  650 = 'Clamp Cylinder A1 Failed to Advance... Check Q1.0...' | German: 'S3 650 Row 66 Failed To Advance.. Check Qxxx.x German' | French: 'S3 650 Row 66 Failed To Advance.. Check Qxxx.x French'
  651 = 'Clamp Cylinder A1 Failed to Return... Check Q1.1...' | German: 'S3 651 Row 66 Failed To Return.. Check Qxxx.x German' | French: 'S3 651 Row 66 Failed To Return.. Check Qxxx.x French'
  652 = 'Clamp Cylinder A1 Lost Advanced... Check I1.0...' | German: 'S3 652 Row 66 Lost Advance Position... Check Ixxx.x German' | French: 'S3 652 Row 66 Lost Advance Position... Check Ixxx.x French'
  653 = 'Clamp Cylinder A1 Lost Returned... Check I1.1...' | German: 'S3 653 Row 66 Lost Return Position... Check Ixxx.x German' | French: 'S3 653 Row 66 Lost Return Position... Check Ixxx.x French'
  654 = 'Clamp Cylinder A1 Switch Fault... Check I1.0, I1.1...' | German: 'S3 654 Row 66 Switch Fault... Check Ixxx.x / Ixxx.x German' | French: 'S3 654 Row 66 Switch Fault... Check Ixxx.x / Ixxx.x French'
  655 = 'Spare' | German: 'S3 655 Row 66 Spare Message German' | French: 'S3 655 Row 66 Spare Message French'
  656 = 'Spare' | German: 'S3 656 Row 66 Spare Message German' | French: 'S3 656 Row 66 Spare Message French'
  657 = 'Spare' | German: 'S3 657 Row 66 Spare Message German' | French: 'S3 657 Row 66 Spare Message French'
  658 = 'Spare' | German: 'S3 658 Row 66 Spare Message German' | French: 'S3 658 Row 66 Spare Message French'
  659 = 'Spare' | German: 'S3 659 Row 66 Spare Message German' | French: 'S3 659 Row 66 Spare Message French'
  660 = 'Clamp Cylinder A1 Failed to Advance... Check Q1.0...' | German: 'S3 660 Row 67 Failed To Advance.. Check Qxxx.x German' | French: 'S3 660 Row 67 Failed To Advance.. Check Qxxx.x French'
  661 = 'Clamp Cylinder A1 Failed to Return... Check Q1.1...' | German: 'S3 661 Row 67 Failed To Return.. Check Qxxx.x German' | French: 'S3 661 Row 67 Failed To Return.. Check Qxxx.x French'
  662 = 'Clamp Cylinder A1 Lost Advanced... Check I1.0...' | German: 'S3 662 Row 67 Lost Advance Position... Check Ixxx.x German' | French: 'S3 662 Row 67 Lost Advance Position... Check Ixxx.x French'
  663 = 'Clamp Cylinder A1 Lost Returned... Check I1.1...' | German: 'S3 663 Row 67 Lost Return Position... Check Ixxx.x German' | French: 'S3 663 Row 67 Lost Return Position... Check Ixxx.x French'
  664 = 'Clamp Cylinder A1 Switch Fault... Check I1.0, I1.1...' | German: 'S3 664 Row 67 Switch Fault... Check Ixxx.x / Ixxx.x German' | French: 'S3 664 Row 67 Switch Fault... Check Ixxx.x / Ixxx.x French'
  665 = 'Spare' | German: 'S3 665 Row 67 Spare Message German' | French: 'S3 665 Row 67 Spare Message French'
  666 = 'Spare' | German: 'S3 666 Row 67 Spare Message German' | French: 'S3 666 Row 67 Spare Message French'
  667 = 'Spare' | German: 'S3 667 Row 67 Spare Message German' | French: 'S3 667 Row 67 Spare Message French'
  668 = 'Spare' | German: 'S3 668 Row 67 Spare Message German' | French: 'S3 668 Row 67 Spare Message French'
  669 = 'Spare' | German: 'S3 669 Row 67 Spare Message German' | French: 'S3 669 Row 67 Spare Message French'
  670 = 'Clamp Cylinder A1 Failed to Advance... Check Q1.0...' | German: 'S3 670 Row 68 Failed To Advance.. Check Qxxx.x German' | French: 'S3 670 Row 68 Failed To Advance.. Check Qxxx.x French'
  671 = 'Clamp Cylinder A1 Failed to Return... Check Q1.1...' | German: 'S3 671 Row 68 Failed To Return.. Check Qxxx.x German' | French: 'S3 671 Row 68 Failed To Return.. Check Qxxx.x French'
  672 = 'Clamp Cylinder A1 Lost Advanced... Check I1.0...' | German: 'S3 672 Row 68 Lost Advance Position... Check Ixxx.x German' | French: 'S3 672 Row 68 Lost Advance Position... Check Ixxx.x French'
  673 = 'Clamp Cylinder A1 Lost Returned... Check I1.1...' | German: 'S3 673 Row 68 Lost Return Position... Check Ixxx.x German' | French: 'S3 673 Row 68 Lost Return Position... Check Ixxx.x French'
  674 = 'Clamp Cylinder A1 Switch Fault... Check I1.0, I1.1...' | German: 'S3 674 Row 68 Switch Fault... Check Ixxx.x / Ixxx.x German' | French: 'S3 674 Row 68 Switch Fault... Check Ixxx.x / Ixxx.x French'
  675 = 'Spare' | German: 'S3 675 Row 68 Spare Message German' | French: 'S3 675 Row 68 Spare Message French'
  676 = 'Spare' | German: 'S3 676 Row 68 Spare Message German' | French: 'S3 676 Row 68 Spare Message French'
  677 = 'Spare' | German: 'S3 677 Row 68 Spare Message German' | French: 'S3 677 Row 68 Spare Message French'
  678 = 'Spare' | German: 'S3 678 Row 68 Spare Message German' | French: 'S3 678 Row 68 Spare Message French'
  679 = 'Spare' | German: 'S3 679 Row 68 Spare Message German' | French: 'S3 679 Row 68 Spare Message French'
  680 = 'Clamp Cylinder A1 Failed to Advance... Check Q1.0...' | German: 'S3 680 Row 69 Failed To Advance.. Check Qxxx.x German' | French: 'S3 680 Row 69 Failed To Advance.. Check Qxxx.x French'
  681 = 'Clamp Cylinder A1 Failed to Return... Check Q1.1...' | German: 'S3 681 Row 69 Failed To Return.. Check Qxxx.x German' | French: 'S3 681 Row 69 Failed To Return.. Check Qxxx.x French'
  682 = 'Clamp Cylinder A1 Lost Advanced... Check I1.0...' | German: 'S3 682 Row 69 Lost Advance Position... Check Ixxx.x German' | French: 'S3 682 Row 69 Lost Advance Position... Check Ixxx.x French'
  683 = 'Clamp Cylinder A1 Lost Returned... Check I1.1...' | German: 'S3 683 Row 69 Lost Return Position... Check Ixxx.x German' | French: 'S3 683 Row 69 Lost Return Position... Check Ixxx.x French'
  684 = 'Clamp Cylinder A1 Switch Fault... Check I1.0, I1.1...' | German: 'S3 684 Row 69 Switch Fault... Check Ixxx.x / Ixxx.x German' | French: 'S3 684 Row 69 Switch Fault... Check Ixxx.x / Ixxx.x French'
  685 = 'Spare' | German: 'S3 685 Row 69 Spare Message German' | French: 'S3 685 Row 69 Spare Message French'
  686 = 'Spare' | German: 'S3 686 Row 69 Spare Message German' | French: 'S3 686 Row 69 Spare Message French'
  687 = 'Spare' | German: 'S3 687 Row 69 Spare Message German' | French: 'S3 687 Row 69 Spare Message French'
  688 = 'Spare' | German: 'S3 688 Row 69 Spare Message German' | French: 'S3 688 Row 69 Spare Message French'
  689 = 'Spare' | German: 'S3 689 Row 69 Spare Message German' | French: 'S3 689 Row 69 Spare Message French'
  690 = 'Clamp Cylinder A1 Failed to Advance... Check Q1.0...' | German: 'S3 690 Row 70 Failed To Advance.. Check Qxxx.x German' | French: 'S3 690 Row 70 Failed To Advance.. Check Qxxx.x French'
  691 = 'Clamp Cylinder A1 Failed to Return... Check Q1.1...' | German: 'S3 691 Row 70 Failed To Return.. Check Qxxx.x German' | French: 'S3 691 Row 70 Failed To Return.. Check Qxxx.x French'
  692 = 'Clamp Cylinder A1 Lost Advanced... Check I1.0...' | German: 'S3 692 Row 70 Lost Advance Position... Check Ixxx.x German' | French: 'S3 692 Row 70 Lost Advance Position... Check Ixxx.x French'
  693 = 'Clamp Cylinder A1 Lost Returned... Check I1.1...' | German: 'S3 693 Row 70 Lost Return Position... Check Ixxx.x German' | French: 'S3 693 Row 70 Lost Return Position... Check Ixxx.x French'
  694 = 'Clamp Cylinder A1 Switch Fault... Check I1.0, I1.1...' | German: 'S3 694 Row 70 Switch Fault... Check Ixxx.x / Ixxx.x German' | French: 'S3 694 Row 70 Switch Fault... Check Ixxx.x / Ixxx.x French'
  695 = 'Spare' | German: 'S3 695 Row 70 Spare Message German' | French: 'S3 695 Row 70 Spare Message French'
  696 = 'Spare' | German: 'S3 696 Row 70 Spare Message German' | French: 'S3 696 Row 70 Spare Message French'
  697 = 'Spare' | German: 'S3 697 Row 70 Spare Message German' | French: 'S3 697 Row 70 Spare Message French'
  698 = 'Spare' | German: 'S3 698 Row 70 Spare Message German' | French: 'S3 698 Row 70 Spare Message French'
  699 = 'Spare' | German: 'S3 699 Row 70 Spare Message German' | French: 'S3 699 Row 70 Spare Message French'
  700 = 'Clamp Cylinder A1 Failed to Advance... Check Q1.0...' | German: 'S3 700 Row 71 Failed To Advance.. Check Qxxx.x German' | French: 'S3 700 Row 71 Failed To Advance.. Check Qxxx.x French'
  701 = 'Clamp Cylinder A1 Failed to Return... Check Q1.1...' | German: 'S3 701 Row 71 Failed To Return.. Check Qxxx.x German' | French: 'S3 701 Row 71 Failed To Return.. Check Qxxx.x French'
  702 = 'Clamp Cylinder A1 Lost Advanced... Check I1.0...' | German: 'S3 702 Row 71 Lost Advance Position... Check Ixxx.x German' | French: 'S3 702 Row 71 Lost Advance Position... Check Ixxx.x French'
  703 = 'Clamp Cylinder A1 Lost Returned... Check I1.1...' | German: 'S3 703 Row 71 Lost Return Position... Check Ixxx.x German' | French: 'S3 703 Row 71 Lost Return Position... Check Ixxx.x French'
  704 = 'Clamp Cylinder A1 Switch Fault... Check I1.0, I1.1...' | German: 'S3 704 Row 71 Switch Fault... Check Ixxx.x / Ixxx.x German' | French: 'S3 704 Row 71 Switch Fault... Check Ixxx.x / Ixxx.x French'
  705 = 'Spare' | German: 'S3 705 Row 71 Spare Message German' | French: 'S3 705 Row 71 Spare Message French'
  706 = 'Spare' | German: 'S3 706 Row 71 Spare Message German' | French: 'S3 706 Row 71 Spare Message French'
  707 = 'Spare' | German: 'S3 707 Row 71 Spare Message German' | French: 'S3 707 Row 71 Spare Message French'
  708 = 'Spare' | German: 'S3 708 Row 71 Spare Message German' | French: 'S3 708 Row 71 Spare Message French'
  709 = 'Spare' | German: 'S3 709 Row 71 Spare Message German' | French: 'S3 709 Row 71 Spare Message French'
  710 = 'Clamp Cylinder A1 Failed to Advance... Check Q1.0...' | German: 'S3 710 Row 72 Failed To Advance.. Check Qxxx.x German' | French: 'S3 710 Row 72 Failed To Advance.. Check Qxxx.x French'
  711 = 'Clamp Cylinder A1 Failed to Return... Check Q1.1...' | German: 'S3 711 Row 72 Failed To Return.. Check Qxxx.x German' | French: 'S3 711 Row 72 Failed To Return.. Check Qxxx.x French'
  712 = 'Clamp Cylinder A1 Lost Advanced... Check I1.0...' | German: 'S3 712 Row 72 Lost Advance Position... Check Ixxx.x German' | French: 'S3 712 Row 72 Lost Advance Position... Check Ixxx.x French'
  713 = 'Clamp Cylinder A1 Lost Returned... Check I1.1...' | German: 'S3 713 Row 72 Lost Return Position... Check Ixxx.x German' | French: 'S3 713 Row 72 Lost Return Position... Check Ixxx.x French'
  714 = 'Clamp Cylinder A1 Switch Fault... Check I1.0, I1.1...' | German: 'S3 714 Row 72 Switch Fault... Check Ixxx.x / Ixxx.x German' | French: 'S3 714 Row 72 Switch Fault... Check Ixxx.x / Ixxx.x French'
  715 = 'Spare' | German: 'S3 715 Row 72 Spare Message German' | French: 'S3 715 Row 72 Spare Message French'
  716 = 'Spare' | German: 'S3 716 Row 72 Spare Message German' | French: 'S3 716 Row 72 Spare Message French'
  717 = 'Spare' | German: 'S3 717 Row 72 Spare Message German' | French: 'S3 717 Row 72 Spare Message French'
  718 = 'Spare' | German: 'S3 718 Row 72 Spare Message German' | French: 'S3 718 Row 72 Spare Message French'
  719 = 'Spare' | German: 'S3 719 Row 72 Spare Message German' | French: 'S3 719 Row 72 Spare Message French'
  720 = 'Clamp Cylinder A1 Failed to Advance... Check Q1.0...' | German: 'S3 720 Row 73 Failed To Advance.. Check Qxxx.x German' | French: 'S3 720 Row 73 Failed To Advance.. Check Qxxx.x French'
  721 = 'Clamp Cylinder A1 Failed to Return... Check Q1.1...' | German: 'S3 721 Row 73 Failed To Return.. Check Qxxx.x German' | French: 'S3 721 Row 73 Failed To Return.. Check Qxxx.x French'
  722 = 'Clamp Cylinder A1 Lost Advanced... Check I1.0...' | German: 'S3 722 Row 73 Lost Advance Position... Check Ixxx.x German' | French: 'S3 722 Row 73 Lost Advance Position... Check Ixxx.x French'
  723 = 'Clamp Cylinder A1 Lost Returned... Check I1.1...' | German: 'S3 723 Row 73 Lost Return Position... Check Ixxx.x German' | French: 'S3 723 Row 73 Lost Return Position... Check Ixxx.x French'
  724 = 'Clamp Cylinder A1 Switch Fault... Check I1.0, I1.1...' | German: 'S3 724 Row 73 Switch Fault... Check Ixxx.x / Ixxx.x German' | French: 'S3 724 Row 73 Switch Fault... Check Ixxx.x / Ixxx.x French'
  725 = 'Spare' | German: 'S3 725 Row 73 Spare Message German' | French: 'S3 725 Row 73 Spare Message French'
  726 = 'Spare' | German: 'S3 726 Row 73 Spare Message German' | French: 'S3 726 Row 73 Spare Message French'
  727 = 'Spare' | German: 'S3 727 Row 73 Spare Message German' | French: 'S3 727 Row 73 Spare Message French'
  728 = 'Spare' | German: 'S3 728 Row 73 Spare Message German' | French: 'S3 728 Row 73 Spare Message French'
  729 = 'Spare' | German: 'S3 729 Row 73 Spare Message German' | French: 'S3 729 Row 73 Spare Message French'
  730 = 'Clamp Cylinder A1 Failed to Advance... Check Q1.0...' | German: 'S3 730 Row 74 Failed To Advance.. Check Qxxx.x German' | French: 'S3 730 Row 74 Failed To Advance.. Check Qxxx.x French'
  731 = 'Clamp Cylinder A1 Failed to Return... Check Q1.1...' | German: 'S3 731 Row 74 Failed To Return.. Check Qxxx.x German' | French: 'S3 731 Row 74 Failed To Return.. Check Qxxx.x French'
  732 = 'Clamp Cylinder A1 Lost Advanced... Check I1.0...' | German: 'S3 732 Row 74 Lost Advance Position... Check Ixxx.x German' | French: 'S3 732 Row 74 Lost Advance Position... Check Ixxx.x French'
  733 = 'Clamp Cylinder A1 Lost Returned... Check I1.1...' | German: 'S3 733 Row 74 Lost Return Position... Check Ixxx.x German' | French: 'S3 733 Row 74 Lost Return Position... Check Ixxx.x French'
  734 = 'Clamp Cylinder A1 Switch Fault... Check I1.0, I1.1...' | German: 'S3 734 Row 74 Switch Fault... Check Ixxx.x / Ixxx.x German' | French: 'S3 734 Row 74 Switch Fault... Check Ixxx.x / Ixxx.x French'
  735 = 'Spare' | German: 'S3 735 Row 74 Spare Message German' | French: 'S3 735 Row 74 Spare Message French'
  736 = 'Spare' | German: 'S3 736 Row 74 Spare Message German' | French: 'S3 736 Row 74 Spare Message French'
  737 = 'Spare' | German: 'S3 737 Row 74 Spare Message German' | French: 'S3 737 Row 74 Spare Message French'
  738 = 'Spare' | German: 'S3 738 Row 74 Spare Message German' | French: 'S3 738 Row 74 Spare Message French'
  739 = 'Spare' | German: 'S3 739 Row 74 Spare Message German' | French: 'S3 739 Row 74 Spare Message French'
  740 = 'Clamp Cylinder A1 Failed to Advance... Check Q1.0...' | German: 'S3 740 Row 75 Failed To Advance.. Check Qxxx.x German' | French: 'S3 740 Row 75 Failed To Advance.. Check Qxxx.x French'
  741 = 'Clamp Cylinder A1 Failed to Return... Check Q1.1...' | German: 'S3 741 Row 75 Failed To Return.. Check Qxxx.x German' | French: 'S3 741 Row 75 Failed To Return.. Check Qxxx.x French'
  742 = 'Clamp Cylinder A1 Lost Advanced... Check I1.0...' | German: 'S3 742 Row 75 Lost Advance Position... Check Ixxx.x German' | French: 'S3 742 Row 75 Lost Advance Position... Check Ixxx.x French'
  743 = 'Clamp Cylinder A1 Lost Returned... Check I1.1...' | German: 'S3 743 Row 75 Lost Return Position... Check Ixxx.x German' | French: 'S3 743 Row 75 Lost Return Position... Check Ixxx.x French'
  744 = 'Clamp Cylinder A1 Switch Fault... Check I1.0, I1.1...' | German: 'S3 744 Row 75 Switch Fault... Check Ixxx.x / Ixxx.x German' | French: 'S3 744 Row 75 Switch Fault... Check Ixxx.x / Ixxx.x French'
  745 = 'Spare' | German: 'S3 745 Row 75 Spare Message German' | French: 'S3 745 Row 75 Spare Message French'
  746 = 'Spare' | German: 'S3 746 Row 75 Spare Message German' | French: 'S3 746 Row 75 Spare Message French'
  747 = 'Spare' | German: 'S3 747 Row 75 Spare Message German' | French: 'S3 747 Row 75 Spare Message French'
  748 = 'Spare' | German: 'S3 748 Row 75 Spare Message German' | French: 'S3 748 Row 75 Spare Message French'
  749 = 'Spare' | German: 'S3 749 Row 75 Spare Message German' | French: 'S3 749 Row 75 Spare Message French'
  750 = 'Clamp Cylinder A1 Failed to Advance... Check Q1.0...' | German: 'S3 750 Row 76 Failed To Advance.. Check Qxxx.x German' | French: 'S3 750 Row 76 Failed To Advance.. Check Qxxx.x French'
  751 = 'Clamp Cylinder A1 Failed to Return... Check Q1.1...' | German: 'S3 751 Row 76 Failed To Return.. Check Qxxx.x German' | French: 'S3 751 Row 76 Failed To Return.. Check Qxxx.x French'
  752 = 'Clamp Cylinder A1 Lost Advanced... Check I1.0...' | German: 'S3 752 Row 76 Lost Advance Position... Check Ixxx.x German' | French: 'S3 752 Row 76 Lost Advance Position... Check Ixxx.x French'
  753 = 'Clamp Cylinder A1 Lost Returned... Check I1.1...' | German: 'S3 753 Row 76 Lost Return Position... Check Ixxx.x German' | French: 'S3 753 Row 76 Lost Return Position... Check Ixxx.x French'
  754 = 'Clamp Cylinder A1 Switch Fault... Check I1.0, I1.1...' | German: 'S3 754 Row 76 Switch Fault... Check Ixxx.x / Ixxx.x German' | French: 'S3 754 Row 76 Switch Fault... Check Ixxx.x / Ixxx.x French'
  755 = 'Spare' | German: 'S3 755 Row 76 Spare Message German' | French: 'S3 755 Row 76 Spare Message French'
  756 = 'Spare' | German: 'S3 756 Row 76 Spare Message German' | French: 'S3 756 Row 76 Spare Message French'
  757 = 'Spare' | German: 'S3 757 Row 76 Spare Message German' | French: 'S3 757 Row 76 Spare Message French'
  758 = 'Spare' | German: 'S3 758 Row 76 Spare Message German' | French: 'S3 758 Row 76 Spare Message French'
  759 = 'Spare' | German: 'S3 759 Row 76 Spare Message German' | French: 'S3 759 Row 76 Spare Message French'
  760 = 'Clamp Cylinder A1 Failed to Advance... Check Q1.0...' | German: 'S3 760 Row 77 Failed To Advance.. Check Qxxx.x German' | French: 'S3 760 Row 77 Failed To Advance.. Check Qxxx.x French'
  761 = 'Clamp Cylinder A1 Failed to Return... Check Q1.1...' | German: 'S3 761 Row 77 Failed To Return.. Check Qxxx.x German' | French: 'S3 761 Row 77 Failed To Return.. Check Qxxx.x French'
  762 = 'Clamp Cylinder A1 Lost Advanced... Check I1.0...' | German: 'S3 762 Row 77 Lost Advance Position... Check Ixxx.x German' | French: 'S3 762 Row 77 Lost Advance Position... Check Ixxx.x French'
  763 = 'Clamp Cylinder A1 Lost Returned... Check I1.1...' | German: 'S3 763 Row 77 Lost Return Position... Check Ixxx.x German' | French: 'S3 763 Row 77 Lost Return Position... Check Ixxx.x French'
  764 = 'Clamp Cylinder A1 Switch Fault... Check I1.0, I1.1...' | German: 'S3 764 Row 77 Switch Fault... Check Ixxx.x / Ixxx.x German' | French: 'S3 764 Row 77 Switch Fault... Check Ixxx.x / Ixxx.x French'
  765 = 'Spare' | German: 'S3 765 Row 77 Spare Message German' | French: 'S3 765 Row 77 Spare Message French'
  766 = 'Spare' | German: 'S3 766 Row 77 Spare Message German' | French: 'S3 766 Row 77 Spare Message French'
  767 = 'Spare' | German: 'S3 767 Row 77 Spare Message German' | French: 'S3 767 Row 77 Spare Message French'
  768 = 'Spare' | German: 'S3 768 Row 77 Spare Message German' | French: 'S3 768 Row 77 Spare Message French'
  769 = 'Spare' | German: 'S3 769 Row 77 Spare Message German' | French: 'S3 769 Row 77 Spare Message French'
  770 = 'Clamp Cylinder A1 Failed to Advance... Check Q1.0...' | German: 'S3 770 Row 78 Failed To Advance.. Check Qxxx.x German' | French: 'S3 770 Row 78 Failed To Advance.. Check Qxxx.x French'
  771 = 'Clamp Cylinder A1 Failed to Return... Check Q1.1...' | German: 'S3 771 Row 78 Failed To Return.. Check Qxxx.x German' | French: 'S3 771 Row 78 Failed To Return.. Check Qxxx.x French'
  772 = 'Clamp Cylinder A1 Lost Advanced... Check I1.0...' | German: 'S3 772 Row 78 Lost Advance Position... Check Ixxx.x German' | French: 'S3 772 Row 78 Lost Advance Position... Check Ixxx.x French'
  773 = 'Clamp Cylinder A1 Lost Returned... Check I1.1...' | German: 'S3 773 Row 78 Lost Return Position... Check Ixxx.x German' | French: 'S3 773 Row 78 Lost Return Position... Check Ixxx.x French'
  774 = 'Clamp Cylinder A1 Switch Fault... Check I1.0, I1.1...' | German: 'S3 774 Row 78 Switch Fault... Check Ixxx.x / Ixxx.x German' | French: 'S3 774 Row 78 Switch Fault... Check Ixxx.x / Ixxx.x French'
  775 = 'Spare' | German: 'S3 775 Row 78 Spare Message German' | French: 'S3 775 Row 78 Spare Message French'
  776 = 'Spare' | German: 'S3 776 Row 78 Spare Message German' | French: 'S3 776 Row 78 Spare Message French'
  777 = 'Spare' | German: 'S3 777 Row 78 Spare Message German' | French: 'S3 777 Row 78 Spare Message French'
  778 = 'Spare' | German: 'S3 778 Row 78 Spare Message German' | French: 'S3 778 Row 78 Spare Message French'
  779 = 'Spare' | German: 'S3 779 Row 78 Spare Message German' | French: 'S3 779 Row 78 Spare Message French'
  780 = 'Clamp Cylinder A1 Failed to Advance... Check Q1.0...' | German: 'S3 780 Row 79 Failed To Advance.. Check Qxxx.x German' | French: 'S3 780 Row 79 Failed To Advance.. Check Qxxx.x French'
  781 = 'Clamp Cylinder A1 Failed to Return... Check Q1.1...' | German: 'S3 781 Row 79 Failed To Return.. Check Qxxx.x German' | French: 'S3 781 Row 79 Failed To Return.. Check Qxxx.x French'
  782 = 'Clamp Cylinder A1 Lost Advanced... Check I1.0...' | German: 'S3 782 Row 79 Lost Advance Position... Check Ixxx.x German' | French: 'S3 782 Row 79 Lost Advance Position... Check Ixxx.x French'
  783 = 'Clamp Cylinder A1 Lost Returned... Check I1.1...' | German: 'S3 783 Row 79 Lost Return Position... Check Ixxx.x German' | French: 'S3 783 Row 79 Lost Return Position... Check Ixxx.x French'
  784 = 'Clamp Cylinder A1 Switch Fault... Check I1.0, I1.1...' | German: 'S3 784 Row 79 Switch Fault... Check Ixxx.x / Ixxx.x German' | French: 'S3 784 Row 79 Switch Fault... Check Ixxx.x / Ixxx.x French'
  785 = 'Spare' | German: 'S3 785 Row 79 Spare Message German' | French: 'S3 785 Row 79 Spare Message French'
  786 = 'Spare' | German: 'S3 786 Row 79 Spare Message German' | French: 'S3 786 Row 79 Spare Message French'
  787 = 'Spare' | German: 'S3 787 Row 79 Spare Message German' | French: 'S3 787 Row 79 Spare Message French'
  788 = 'Spare' | German: 'S3 788 Row 79 Spare Message German' | French: 'S3 788 Row 79 Spare Message French'
  789 = 'Spare' | German: 'S3 789 Row 79 Spare Message German' | French: 'S3 789 Row 79 Spare Message French'
  790 = 'Clamp Cylinder A1 Failed to Advance... Check Q1.0...' | German: 'S3 790 Row 80 Failed To Advance.. Check Qxxx.x German' | French: 'S3 790 Row 80 Failed To Advance.. Check Qxxx.x French'
  791 = 'Clamp Cylinder A1 Failed to Return... Check Q1.1...' | German: 'S3 791 Row 80 Failed To Return.. Check Qxxx.x German' | French: 'S3 791 Row 80 Failed To Return.. Check Qxxx.x French'
  792 = 'Clamp Cylinder A1 Lost Advanced... Check I1.0...' | German: 'S3 792 Row 80 Lost Advance Position... Check Ixxx.x German' | French: 'S3 792 Row 80 Lost Advance Position... Check Ixxx.x French'
  793 = 'Clamp Cylinder A1 Lost Returned... Check I1.1...' | German: 'S3 793 Row 80 Lost Return Position... Check Ixxx.x German' | French: 'S3 793 Row 80 Lost Return Position... Check Ixxx.x French'
  794 = 'Clamp Cylinder A1 Switch Fault... Check I1.0, I1.1...' | German: 'S3 794 Row 80 Switch Fault... Check Ixxx.x / Ixxx.x German' | French: 'S3 794 Row 80 Switch Fault... Check Ixxx.x / Ixxx.x French'
  795 = 'Spare' | German: 'S3 795 Row 80 Spare Message German' | French: 'S3 795 Row 80 Spare Message French'
  796 = 'Spare' | German: 'S3 796 Row 80 Spare Message German' | French: 'S3 796 Row 80 Spare Message French'
  797 = 'Spare' | German: 'S3 797 Row 80 Spare Message German' | French: 'S3 797 Row 80 Spare Message French'
  798 = 'Spare' | German: 'S3 798 Row 80 Spare Message German' | French: 'S3 798 Row 80 Spare Message French'
  799 = 'Spare' | German: 'S3 799 Row 80 Spare Message German' | French: 'S3 799 Row 80 Spare Message French'
  800 = 'Clamp Cylinder A1 Failed to Advance... Check Q1.0...' | German: 'S3 800 Row 81 Failed To Advance.. Check Qxxx.x German' | French: 'S3 800 Row 81 Failed To Advance.. Check Qxxx.x French'
  801 = 'Clamp Cylinder A1 Failed to Return... Check Q1.1...' | German: 'S3 801 Row 81 Failed To Return.. Check Qxxx.x German' | French: 'S3 801 Row 81 Failed To Return.. Check Qxxx.x French'
  802 = 'Clamp Cylinder A1 Lost Advanced... Check I1.0...' | German: 'S3 802 Row 81 Lost Advance Position... Check Ixxx.x German' | French: 'S3 802 Row 81 Lost Advance Position... Check Ixxx.x French'
  803 = 'Clamp Cylinder A1 Lost Returned... Check I1.1...' | German: 'S3 803 Row 81 Lost Return Position... Check Ixxx.x German' | French: 'S3 803 Row 81 Lost Return Position... Check Ixxx.x French'
  804 = 'Clamp Cylinder A1 Switch Fault... Check I1.0, I1.1...' | German: 'S3 804 Row 81 Switch Fault... Check Ixxx.x / Ixxx.x German' | French: 'S3 804 Row 81 Switch Fault... Check Ixxx.x / Ixxx.x French'
  805 = 'Spare' | German: 'S3 805 Row 81 Spare Message German' | French: 'S3 805 Row 81 Spare Message French'
  806 = 'Spare' | German: 'S3 806 Row 81 Spare Message German' | French: 'S3 806 Row 81 Spare Message French'
  807 = 'Spare' | German: 'S3 807 Row 81 Spare Message German' | French: 'S3 807 Row 81 Spare Message French'
  808 = 'Spare' | German: 'S3 808 Row 81 Spare Message German' | French: 'S3 808 Row 81 Spare Message French'
  809 = 'Spare' | German: 'S3 809 Row 81 Spare Message German' | French: 'S3 809 Row 81 Spare Message French'
  810 = 'Clamp Cylinder A1 Failed to Advance... Check Q1.0...' | German: 'S3 810 Row 82 Failed To Advance.. Check Qxxx.x German' | French: 'S3 810 Row 82 Failed To Advance.. Check Qxxx.x French'
  811 = 'Clamp Cylinder A1 Failed to Return... Check Q1.1...' | German: 'S3 811 Row 82 Failed To Return.. Check Qxxx.x German' | French: 'S3 811 Row 82 Failed To Return.. Check Qxxx.x French'
  812 = 'Clamp Cylinder A1 Lost Advanced... Check I1.0...' | German: 'S3 812 Row 82 Lost Advance Position... Check Ixxx.x German' | French: 'S3 812 Row 82 Lost Advance Position... Check Ixxx.x French'
  813 = 'Clamp Cylinder A1 Lost Returned... Check I1.1...' | German: 'S3 813 Row 82 Lost Return Position... Check Ixxx.x German' | French: 'S3 813 Row 82 Lost Return Position... Check Ixxx.x French'
  814 = 'Clamp Cylinder A1 Switch Fault... Check I1.0, I1.1...' | German: 'S3 814 Row 82 Switch Fault... Check Ixxx.x / Ixxx.x German' | French: 'S3 814 Row 82 Switch Fault... Check Ixxx.x / Ixxx.x French'
  815 = 'Spare' | German: 'S3 815 Row 82 Spare Message German' | French: 'S3 815 Row 82 Spare Message French'
  816 = 'Spare' | German: 'S3 816 Row 82 Spare Message German' | French: 'S3 816 Row 82 Spare Message French'
  817 = 'Spare' | German: 'S3 817 Row 82 Spare Message German' | French: 'S3 817 Row 82 Spare Message French'
  818 = 'Spare' | German: 'S3 818 Row 82 Spare Message German' | French: 'S3 818 Row 82 Spare Message French'
  819 = 'Spare' | German: 'S3 819 Row 82 Spare Message German' | French: 'S3 819 Row 82 Spare Message French'
  820 = 'Clamp Cylinder A1 Failed to Advance... Check Q1.0...' | German: 'S3 820 Row 83 Failed To Advance.. Check Qxxx.x German' | French: 'S3 820 Row 83 Failed To Advance.. Check Qxxx.x French'
  821 = 'Clamp Cylinder A1 Failed to Return... Check Q1.1...' | German: 'S3 821 Row 83 Failed To Return.. Check Qxxx.x German' | French: 'S3 821 Row 83 Failed To Return.. Check Qxxx.x French'
  822 = 'Clamp Cylinder A1 Lost Advanced... Check I1.0...' | German: 'S3 822 Row 83 Lost Advance Position... Check Ixxx.x German' | French: 'S3 822 Row 83 Lost Advance Position... Check Ixxx.x French'
  823 = 'Clamp Cylinder A1 Lost Returned... Check I1.1...' | German: 'S3 823 Row 83 Lost Return Position... Check Ixxx.x German' | French: 'S3 823 Row 83 Lost Return Position... Check Ixxx.x French'
  824 = 'Clamp Cylinder A1 Switch Fault... Check I1.0, I1.1...' | German: 'S3 824 Row 83 Switch Fault... Check Ixxx.x / Ixxx.x German' | French: 'S3 824 Row 83 Switch Fault... Check Ixxx.x / Ixxx.x French'
  825 = 'Spare' | German: 'S3 825 Row 83 Spare Message German' | French: 'S3 825 Row 83 Spare Message French'
  826 = 'Spare' | German: 'S3 826 Row 83 Spare Message German' | French: 'S3 826 Row 83 Spare Message French'
  827 = 'Spare' | German: 'S3 827 Row 83 Spare Message German' | French: 'S3 827 Row 83 Spare Message French'
  828 = 'Spare' | German: 'S3 828 Row 83 Spare Message German' | French: 'S3 828 Row 83 Spare Message French'
  829 = 'Spare' | German: 'S3 829 Row 83 Spare Message German' | French: 'S3 829 Row 83 Spare Message French'
  830 = 'Clamp Cylinder A1 Failed to Advance... Check Q1.0...' | German: 'S3 830 Row 84 Failed To Advance.. Check Qxxx.x German' | French: 'S3 830 Row 84 Failed To Advance.. Check Qxxx.x French'
  831 = 'Clamp Cylinder A1 Failed to Return... Check Q1.1...' | German: 'S3 831 Row 84 Failed To Return.. Check Qxxx.x German' | French: 'S3 831 Row 84 Failed To Return.. Check Qxxx.x French'
  832 = 'Clamp Cylinder A1 Lost Advanced... Check I1.0...' | German: 'S3 832 Row 84 Lost Advance Position... Check Ixxx.x German' | French: 'S3 832 Row 84 Lost Advance Position... Check Ixxx.x French'
  833 = 'Clamp Cylinder A1 Lost Returned... Check I1.1...' | German: 'S3 833 Row 84 Lost Return Position... Check Ixxx.x German' | French: 'S3 833 Row 84 Lost Return Position... Check Ixxx.x French'
  834 = 'Clamp Cylinder A1 Switch Fault... Check I1.0, I1.1...' | German: 'S3 834 Row 84 Switch Fault... Check Ixxx.x / Ixxx.x German' | French: 'S3 834 Row 84 Switch Fault... Check Ixxx.x / Ixxx.x French'
  835 = 'Spare' | German: 'S3 835 Row 84 Spare Message German' | French: 'S3 835 Row 84 Spare Message French'
  836 = 'Spare' | German: 'S3 836 Row 84 Spare Message German' | French: 'S3 836 Row 84 Spare Message French'
  837 = 'Spare' | German: 'S3 837 Row 84 Spare Message German' | French: 'S3 837 Row 84 Spare Message French'
  838 = 'Spare' | German: 'S3 838 Row 84 Spare Message German' | French: 'S3 838 Row 84 Spare Message French'
  839 = 'Spare' | German: 'S3 839 Row 84 Spare Message German' | French: 'S3 839 Row 84 Spare Message French'
  840 = 'Clamp Cylinder A1 Failed to Advance... Check Q1.0...' | German: 'S3 840 Row 85 Failed To Advance.. Check Qxxx.x German' | French: 'S3 840 Row 85 Failed To Advance.. Check Qxxx.x French'
  841 = 'Clamp Cylinder A1 Failed to Return... Check Q1.1...' | German: 'S3 841 Row 85 Failed To Return.. Check Qxxx.x German' | French: 'S3 841 Row 85 Failed To Return.. Check Qxxx.x French'
  842 = 'Clamp Cylinder A1 Lost Advanced... Check I1.0...' | German: 'S3 842 Row 85 Lost Advance Position... Check Ixxx.x German' | French: 'S3 842 Row 85 Lost Advance Position... Check Ixxx.x French'
  843 = 'Clamp Cylinder A1 Lost Returned... Check I1.1...' | German: 'S3 843 Row 85 Lost Return Position... Check Ixxx.x German' | French: 'S3 843 Row 85 Lost Return Position... Check Ixxx.x French'
  844 = 'Clamp Cylinder A1 Switch Fault... Check I1.0, I1.1...' | German: 'S3 844 Row 85 Switch Fault... Check Ixxx.x / Ixxx.x German' | French: 'S3 844 Row 85 Switch Fault... Check Ixxx.x / Ixxx.x French'
  845 = 'Spare' | German: 'S3 845 Row 85 Spare Message German' | French: 'S3 845 Row 85 Spare Message French'
  846 = 'Spare' | German: 'S3 846 Row 85 Spare Message German' | French: 'S3 846 Row 85 Spare Message French'
  847 = 'Spare' | German: 'S3 847 Row 85 Spare Message German' | French: 'S3 847 Row 85 Spare Message French'
  848 = 'Spare' | German: 'S3 848 Row 85 Spare Message German' | French: 'S3 848 Row 85 Spare Message French'
  849 = 'Spare' | German: 'S3 849 Row 85 Spare Message German' | French: 'S3 849 Row 85 Spare Message French'
  850 = 'Clamp Cylinder A1 Failed to Advance... Check Q1.0...' | German: 'S3 850 Row 86 Failed To Advance.. Check Qxxx.x German' | French: 'S3 850 Row 86 Failed To Advance.. Check Qxxx.x French'
  851 = 'Clamp Cylinder A1 Failed to Return... Check Q1.1...' | German: 'S3 851 Row 86 Failed To Return.. Check Qxxx.x German' | French: 'S3 851 Row 86 Failed To Return.. Check Qxxx.x French'
  852 = 'Clamp Cylinder A1 Lost Advanced... Check I1.0...' | German: 'S3 852 Row 86 Lost Advance Position... Check Ixxx.x German' | French: 'S3 852 Row 86 Lost Advance Position... Check Ixxx.x French'
  853 = 'Clamp Cylinder A1 Lost Returned... Check I1.1...' | German: 'S3 853 Row 86 Lost Return Position... Check Ixxx.x German' | French: 'S3 853 Row 86 Lost Return Position... Check Ixxx.x French'
  854 = 'Clamp Cylinder A1 Switch Fault... Check I1.0, I1.1...' | German: 'S3 854 Row 86 Switch Fault... Check Ixxx.x / Ixxx.x German' | French: 'S3 854 Row 86 Switch Fault... Check Ixxx.x / Ixxx.x French'
  855 = 'Spare' | German: 'S3 855 Row 86 Spare Message German' | French: 'S3 855 Row 86 Spare Message French'
  856 = 'Spare' | German: 'S3 856 Row 86 Spare Message German' | French: 'S3 856 Row 86 Spare Message French'
  857 = 'Spare' | German: 'S3 857 Row 86 Spare Message German' | French: 'S3 857 Row 86 Spare Message French'
  858 = 'Spare' | German: 'S3 858 Row 86 Spare Message German' | French: 'S3 858 Row 86 Spare Message French'
  859 = 'Spare' | German: 'S3 859 Row 86 Spare Message German' | French: 'S3 859 Row 86 Spare Message French'
  860 = 'Clamp Cylinder A1 Failed to Advance... Check Q1.0...' | German: 'S3 860 Row 87 Failed To Advance.. Check Qxxx.x German' | French: 'S3 860 Row 87 Failed To Advance.. Check Qxxx.x French'
  861 = 'Clamp Cylinder A1 Failed to Return... Check Q1.1...' | German: 'S3 861 Row 87 Failed To Return.. Check Qxxx.x German' | French: 'S3 861 Row 87 Failed To Return.. Check Qxxx.x French'
  862 = 'Clamp Cylinder A1 Lost Advanced... Check I1.0...' | German: 'S3 862 Row 87 Lost Advance Position... Check Ixxx.x German' | French: 'S3 862 Row 87 Lost Advance Position... Check Ixxx.x French'
  863 = 'Clamp Cylinder A1 Lost Returned... Check I1.1...' | German: 'S3 863 Row 87 Lost Return Position... Check Ixxx.x German' | French: 'S3 863 Row 87 Lost Return Position... Check Ixxx.x French'
  864 = 'Clamp Cylinder A1 Switch Fault... Check I1.0, I1.1...' | German: 'S3 864 Row 87 Switch Fault... Check Ixxx.x / Ixxx.x German' | French: 'S3 864 Row 87 Switch Fault... Check Ixxx.x / Ixxx.x French'
  865 = 'Spare' | German: 'S3 865 Row 87 Spare Message German' | French: 'S3 865 Row 87 Spare Message French'
  866 = 'Spare' | German: 'S3 866 Row 87 Spare Message German' | French: 'S3 866 Row 87 Spare Message French'
  867 = 'Spare' | German: 'S3 867 Row 87 Spare Message German' | French: 'S3 867 Row 87 Spare Message French'
  868 = 'Spare' | German: 'S3 868 Row 87 Spare Message German' | French: 'S3 868 Row 87 Spare Message French'
  869 = 'Spare' | German: 'S3 869 Row 87 Spare Message German' | French: 'S3 869 Row 87 Spare Message French'
  870 = 'Clamp Cylinder A1 Failed to Advance... Check Q1.0...' | German: 'S3 870 Row 88 Failed To Advance.. Check Qxxx.x German' | French: 'S3 870 Row 88 Failed To Advance.. Check Qxxx.x French'
  871 = 'Clamp Cylinder A1 Failed to Return... Check Q1.1...' | German: 'S3 871 Row 88 Failed To Return.. Check Qxxx.x German' | French: 'S3 871 Row 88 Failed To Return.. Check Qxxx.x French'
  872 = 'Clamp Cylinder A1 Lost Advanced... Check I1.0...' | German: 'S3 872 Row 88 Lost Advance Position... Check Ixxx.x German' | French: 'S3 872 Row 88 Lost Advance Position... Check Ixxx.x French'
  873 = 'Clamp Cylinder A1 Lost Returned... Check I1.1...' | German: 'S3 873 Row 88 Lost Return Position... Check Ixxx.x German' | French: 'S3 873 Row 88 Lost Return Position... Check Ixxx.x French'
  874 = 'Clamp Cylinder A1 Switch Fault... Check I1.0, I1.1...' | German: 'S3 874 Row 88 Switch Fault... Check Ixxx.x / Ixxx.x German' | French: 'S3 874 Row 88 Switch Fault... Check Ixxx.x / Ixxx.x French'
  875 = 'Spare' | German: 'S3 875 Row 88 Spare Message German' | French: 'S3 875 Row 88 Spare Message French'
  876 = 'Spare' | German: 'S3 876 Row 88 Spare Message German' | French: 'S3 876 Row 88 Spare Message French'
  877 = 'Spare' | German: 'S3 877 Row 88 Spare Message German' | French: 'S3 877 Row 88 Spare Message French'
  878 = 'Spare' | German: 'S3 878 Row 88 Spare Message German' | French: 'S3 878 Row 88 Spare Message French'
  879 = 'Spare' | German: 'S3 879 Row 88 Spare Message German' | French: 'S3 879 Row 88 Spare Message French'
  880 = 'Clamp Cylinder A1 Failed to Advance... Check Q1.0...' | German: 'S3 880 Row 89 Failed To Advance.. Check Qxxx.x German' | French: 'S3 880 Row 89 Failed To Advance.. Check Qxxx.x French'
  881 = 'Clamp Cylinder A1 Failed to Return... Check Q1.1...' | German: 'S3 881 Row 89 Failed To Return.. Check Qxxx.x German' | French: 'S3 881 Row 89 Failed To Return.. Check Qxxx.x French'
  882 = 'Clamp Cylinder A1 Lost Advanced... Check I1.0...' | German: 'S3 882 Row 89 Lost Advance Position... Check Ixxx.x German' | French: 'S3 882 Row 89 Lost Advance Position... Check Ixxx.x French'
  883 = 'Clamp Cylinder A1 Lost Returned... Check I1.1...' | German: 'S3 883 Row 89 Lost Return Position... Check Ixxx.x German' | French: 'S3 883 Row 89 Lost Return Position... Check Ixxx.x French'
  884 = 'Clamp Cylinder A1 Switch Fault... Check I1.0, I1.1...' | German: 'S3 884 Row 89 Switch Fault... Check Ixxx.x / Ixxx.x German' | French: 'S3 884 Row 89 Switch Fault... Check Ixxx.x / Ixxx.x French'
  885 = 'Spare' | German: 'S3 885 Row 89 Spare Message German' | French: 'S3 885 Row 89 Spare Message French'
  886 = 'Spare' | German: 'S3 886 Row 89 Spare Message German' | French: 'S3 886 Row 89 Spare Message French'
  887 = 'Spare' | German: 'S3 887 Row 89 Spare Message German' | French: 'S3 887 Row 89 Spare Message French'
  888 = 'Spare' | German: 'S3 888 Row 89 Spare Message German' | French: 'S3 888 Row 89 Spare Message French'
  889 = 'Spare' | German: 'S3 889 Row 89 Spare Message German' | French: 'S3 889 Row 89 Spare Message French'
  890 = 'Clamp Cylinder A1 Failed to Advance... Check Q1.0...' | German: 'S3 890 Row 90 Failed To Advance.. Check Qxxx.x German' | French: 'S3 890 Row 90 Failed To Advance.. Check Qxxx.x French'
  891 = 'Clamp Cylinder A1 Failed to Return... Check Q1.1...' | German: 'S3 891 Row 90 Failed To Return.. Check Qxxx.x German' | French: 'S3 891 Row 90 Failed To Return.. Check Qxxx.x French'
  892 = 'Clamp Cylinder A1 Lost Advanced... Check I1.0...' | German: 'S3 892 Row 90 Lost Advance Position... Check Ixxx.x German' | French: 'S3 892 Row 90 Lost Advance Position... Check Ixxx.x French'
  893 = 'Clamp Cylinder A1 Lost Returned... Check I1.1...' | German: 'S3 893 Row 90 Lost Return Position... Check Ixxx.x German' | French: 'S3 893 Row 90 Lost Return Position... Check Ixxx.x French'
  894 = 'Clamp Cylinder A1 Switch Fault... Check I1.0, I1.1...' | German: 'S3 894 Row 90 Switch Fault... Check Ixxx.x / Ixxx.x German' | French: 'S3 894 Row 90 Switch Fault... Check Ixxx.x / Ixxx.x French'
  895 = 'Spare' | German: 'S3 895 Row 90 Spare Message German' | French: 'S3 895 Row 90 Spare Message French'
  896 = 'Spare' | German: 'S3 896 Row 90 Spare Message German' | French: 'S3 896 Row 90 Spare Message French'
  897 = 'Spare' | German: 'S3 897 Row 90 Spare Message German' | French: 'S3 897 Row 90 Spare Message French'
  898 = 'Spare' | German: 'S3 898 Row 90 Spare Message German' | French: 'S3 898 Row 90 Spare Message French'
  899 = 'Spare' | German: 'S3 899 Row 90 Spare Message German' | French: 'S3 899 Row 90 Spare Message French'
  900 = 'Clamp Cylinder A1 Failed to Advance... Check Q1.0...' | German: 'S3 900 Row 91 Failed To Advance.. Check Qxxx.x German' | French: 'S3 900 Row 91 Failed To Advance.. Check Qxxx.x French'
  901 = 'Clamp Cylinder A1 Failed to Return... Check Q1.1...' | German: 'S3 901 Row 91 Failed To Return.. Check Qxxx.x German' | French: 'S3 901 Row 91 Failed To Return.. Check Qxxx.x French'
  902 = 'Clamp Cylinder A1 Lost Advanced... Check I1.0...' | German: 'S3 902 Row 91 Lost Advance Position... Check Ixxx.x German' | French: 'S3 902 Row 91 Lost Advance Position... Check Ixxx.x French'
  903 = 'Clamp Cylinder A1 Lost Returned... Check I1.1...' | German: 'S3 903 Row 91 Lost Return Position... Check Ixxx.x German' | French: 'S3 903 Row 91 Lost Return Position... Check Ixxx.x French'
  904 = 'Clamp Cylinder A1 Switch Fault... Check I1.0, I1.1...' | German: 'S3 904 Row 91 Switch Fault... Check Ixxx.x / Ixxx.x German' | French: 'S3 904 Row 91 Switch Fault... Check Ixxx.x / Ixxx.x French'
  905 = 'Spare' | German: 'S3 905 Row 91 Spare Message German' | French: 'S3 905 Row 91 Spare Message French'
  906 = 'Spare' | German: 'S3 906 Row 91 Spare Message German' | French: 'S3 906 Row 91 Spare Message French'
  907 = 'Spare' | German: 'S3 907 Row 91 Spare Message German' | French: 'S3 907 Row 91 Spare Message French'
  908 = 'Spare' | German: 'S3 908 Row 91 Spare Message German' | French: 'S3 908 Row 91 Spare Message French'
  909 = 'Spare' | German: 'S3 909 Row 91 Spare Message German' | French: 'S3 909 Row 91 Spare Message French'
  910 = 'Clamp Cylinder A1 Failed to Advance... Check Q1.0...' | German: 'S3 910 Row 92 Failed To Advance.. Check Qxxx.x German' | French: 'S3 910 Row 92 Failed To Advance.. Check Qxxx.x French'
  911 = 'Clamp Cylinder A1 Failed to Return... Check Q1.1...' | German: 'S3 911 Row 92 Failed To Return.. Check Qxxx.x German' | French: 'S3 911 Row 92 Failed To Return.. Check Qxxx.x French'
  912 = 'Clamp Cylinder A1 Lost Advanced... Check I1.0...' | German: 'S3 912 Row 92 Lost Advance Position... Check Ixxx.x German' | French: 'S3 912 Row 92 Lost Advance Position... Check Ixxx.x French'
  913 = 'Clamp Cylinder A1 Lost Returned... Check I1.1...' | German: 'S3 913 Row 92 Lost Return Position... Check Ixxx.x German' | French: 'S3 913 Row 92 Lost Return Position... Check Ixxx.x French'
  914 = 'Clamp Cylinder A1 Switch Fault... Check I1.0, I1.1...' | German: 'S3 914 Row 92 Switch Fault... Check Ixxx.x / Ixxx.x German' | French: 'S3 914 Row 92 Switch Fault... Check Ixxx.x / Ixxx.x French'
  915 = 'Spare' | German: 'S3 915 Row 92 Spare Message German' | French: 'S3 915 Row 92 Spare Message French'
  916 = 'Spare' | German: 'S3 916 Row 92 Spare Message German' | French: 'S3 916 Row 92 Spare Message French'
  917 = 'Spare' | German: 'S3 917 Row 92 Spare Message German' | French: 'S3 917 Row 92 Spare Message French'
  918 = 'Spare' | German: 'S3 918 Row 92 Spare Message German' | French: 'S3 918 Row 92 Spare Message French'
  919 = 'Spare' | German: 'S3 919 Row 92 Spare Message German' | French: 'S3 919 Row 92 Spare Message French'
  920 = 'Clamp Cylinder A1 Failed to Advance... Check Q1.0...' | German: 'S3 920 Row 93 Failed To Advance.. Check Qxxx.x German' | French: 'S3 920 Row 93 Failed To Advance.. Check Qxxx.x French'
  921 = 'Clamp Cylinder A1 Failed to Return... Check Q1.1...' | German: 'S3 921 Row 93 Failed To Return.. Check Qxxx.x German' | French: 'S3 921 Row 93 Failed To Return.. Check Qxxx.x French'
  922 = 'Clamp Cylinder A1 Lost Advanced... Check I1.0...' | German: 'S3 922 Row 93 Lost Advance Position... Check Ixxx.x German' | French: 'S3 922 Row 93 Lost Advance Position... Check Ixxx.x French'
  923 = 'Clamp Cylinder A1 Lost Returned... Check I1.1...' | German: 'S3 923 Row 93 Lost Return Position... Check Ixxx.x German' | French: 'S3 923 Row 93 Lost Return Position... Check Ixxx.x French'
  924 = 'Clamp Cylinder A1 Switch Fault... Check I1.0, I1.1...' | German: 'S3 924 Row 93 Switch Fault... Check Ixxx.x / Ixxx.x German' | French: 'S3 924 Row 93 Switch Fault... Check Ixxx.x / Ixxx.x French'
  925 = 'Spare' | German: 'S3 925 Row 93 Spare Message German' | French: 'S3 925 Row 93 Spare Message French'
  926 = 'Spare' | German: 'S3 926 Row 93 Spare Message German' | French: 'S3 926 Row 93 Spare Message French'
  927 = 'Spare' | German: 'S3 927 Row 93 Spare Message German' | French: 'S3 927 Row 93 Spare Message French'
  928 = 'Spare' | German: 'S3 928 Row 93 Spare Message German' | French: 'S3 928 Row 93 Spare Message French'
  929 = 'Spare' | German: 'S3 929 Row 93 Spare Message German' | French: 'S3 929 Row 93 Spare Message French'
  930 = 'Clamp Cylinder A1 Failed to Advance... Check Q1.0...' | German: 'S3 930 Row 94 Failed To Advance.. Check Qxxx.x German' | French: 'S3 930 Row 94 Failed To Advance.. Check Qxxx.x French'
  931 = 'Clamp Cylinder A1 Failed to Return... Check Q1.1...' | German: 'S3 931 Row 94 Failed To Return.. Check Qxxx.x German' | French: 'S3 931 Row 94 Failed To Return.. Check Qxxx.x French'
  932 = 'Clamp Cylinder A1 Lost Advanced... Check I1.0...' | German: 'S3 932 Row 94 Lost Advance Position... Check Ixxx.x German' | French: 'S3 932 Row 94 Lost Advance Position... Check Ixxx.x French'
  933 = 'Clamp Cylinder A1 Lost Returned... Check I1.1...' | German: 'S3 933 Row 94 Lost Return Position... Check Ixxx.x German' | French: 'S3 933 Row 94 Lost Return Position... Check Ixxx.x French'
  934 = 'Clamp Cylinder A1 Switch Fault... Check I1.0, I1.1...' | German: 'S3 934 Row 94 Switch Fault... Check Ixxx.x / Ixxx.x German' | French: 'S3 934 Row 94 Switch Fault... Check Ixxx.x / Ixxx.x French'
  935 = 'Spare' | German: 'S3 935 Row 94 Spare Message German' | French: 'S3 935 Row 94 Spare Message French'
  936 = 'Spare' | German: 'S3 936 Row 94 Spare Message German' | French: 'S3 936 Row 94 Spare Message French'
  937 = 'Spare' | German: 'S3 937 Row 94 Spare Message German' | French: 'S3 937 Row 94 Spare Message French'
  938 = 'Spare' | German: 'S3 938 Row 94 Spare Message German' | French: 'S3 938 Row 94 Spare Message French'
  939 = 'Spare' | German: 'S3 939 Row 94 Spare Message German' | French: 'S3 939 Row 94 Spare Message French'
  940 = 'Clamp Cylinder A1 Failed to Advance... Check Q1.0...' | German: 'S3 940 Row 95 Failed To Advance.. Check Qxxx.x German' | French: 'S3 940 Row 95 Failed To Advance.. Check Qxxx.x French'
  941 = 'Clamp Cylinder A1 Failed to Return... Check Q1.1...' | German: 'S3 941 Row 95 Failed To Return.. Check Qxxx.x German' | French: 'S3 941 Row 95 Failed To Return.. Check Qxxx.x French'
  942 = 'Clamp Cylinder A1 Lost Advanced... Check I1.0...' | German: 'S3 942 Row 95 Lost Advance Position... Check Ixxx.x German' | French: 'S3 942 Row 95 Lost Advance Position... Check Ixxx.x French'
  943 = 'Clamp Cylinder A1 Lost Returned... Check I1.1...' | German: 'S3 943 Row 95 Lost Return Position... Check Ixxx.x German' | French: 'S3 943 Row 95 Lost Return Position... Check Ixxx.x French'
  944 = 'Clamp Cylinder A1 Switch Fault... Check I1.0, I1.1...' | German: 'S3 944 Row 95 Switch Fault... Check Ixxx.x / Ixxx.x German' | French: 'S3 944 Row 95 Switch Fault... Check Ixxx.x / Ixxx.x French'
  945 = 'Spare' | German: 'S3 945 Row 95 Spare Message German' | French: 'S3 945 Row 95 Spare Message French'
  946 = 'Spare' | German: 'S3 946 Row 95 Spare Message German' | French: 'S3 946 Row 95 Spare Message French'
  947 = 'Spare' | German: 'S3 947 Row 95 Spare Message German' | French: 'S3 947 Row 95 Spare Message French'
  948 = 'Spare' | German: 'S3 948 Row 95 Spare Message German' | French: 'S3 948 Row 95 Spare Message French'
  949 = 'Spare' | German: 'S3 949 Row 95 Spare Message German' | French: 'S3 949 Row 95 Spare Message French'
  950 = 'Clamp Cylinder A1 Failed to Advance... Check Q1.0...' | German: 'S3 950 Row 96 Failed To Advance.. Check Qxxx.x German' | French: 'S3 950 Row 96 Failed To Advance.. Check Qxxx.x French'
  951 = 'Clamp Cylinder A1 Failed to Return... Check Q1.1...' | German: 'S3 951 Row 96 Failed To Return.. Check Qxxx.x German' | French: 'S3 951 Row 96 Failed To Return.. Check Qxxx.x French'
  952 = 'Clamp Cylinder A1 Lost Advanced... Check I1.0...' | German: 'S3 952 Row 96 Lost Advance Position... Check Ixxx.x German' | French: 'S3 952 Row 96 Lost Advance Position... Check Ixxx.x French'
  953 = 'Clamp Cylinder A1 Lost Returned... Check I1.1...' | German: 'S3 953 Row 96 Lost Return Position... Check Ixxx.x German' | French: 'S3 953 Row 96 Lost Return Position... Check Ixxx.x French'
  954 = 'Clamp Cylinder A1 Switch Fault... Check I1.0, I1.1...' | German: 'S3 954 Row 96 Switch Fault... Check Ixxx.x / Ixxx.x German' | French: 'S3 954 Row 96 Switch Fault... Check Ixxx.x / Ixxx.x French'
  955 = 'Spare' | German: 'S3 955 Row 96 Spare Message German' | French: 'S3 955 Row 96 Spare Message French'
  956 = 'Spare' | German: 'S3 956 Row 96 Spare Message German' | French: 'S3 956 Row 96 Spare Message French'
  957 = 'Spare' | German: 'S3 957 Row 96 Spare Message German' | French: 'S3 957 Row 96 Spare Message French'
  958 = 'Spare' | German: 'S3 958 Row 96 Spare Message German' | French: 'S3 958 Row 96 Spare Message French'
  959 = 'Spare' | German: 'S3 959 Row 96 Spare Message German' | French: 'S3 959 Row 96 Spare Message French'
  960 = 'Clamp Cylinder A1 Failed to Advance... Check Q1.0...' | German: 'S3 960 Row 97 Failed To Advance.. Check Qxxx.x German' | French: 'S3 960 Row 97 Failed To Advance.. Check Qxxx.x French'
  961 = 'Clamp Cylinder A1 Failed to Return... Check Q1.1...' | German: 'S3 961 Row 97 Failed To Return.. Check Qxxx.x German' | French: 'S3 961 Row 97 Failed To Return.. Check Qxxx.x French'
  962 = 'Clamp Cylinder A1 Lost Advanced... Check I1.0...' | German: 'S3 962 Row 97 Lost Advance Position... Check Ixxx.x German' | French: 'S3 962 Row 97 Lost Advance Position... Check Ixxx.x French'
  963 = 'Clamp Cylinder A1 Lost Returned... Check I1.1...' | German: 'S3 963 Row 97 Lost Return Position... Check Ixxx.x German' | French: 'S3 963 Row 97 Lost Return Position... Check Ixxx.x French'
  964 = 'Clamp Cylinder A1 Switch Fault... Check I1.0, I1.1...' | German: 'S3 964 Row 97 Switch Fault... Check Ixxx.x / Ixxx.x German' | French: 'S3 964 Row 97 Switch Fault... Check Ixxx.x / Ixxx.x French'
  965 = 'Spare' | German: 'S3 965 Row 97 Spare Message German' | French: 'S3 965 Row 97 Spare Message French'
  966 = 'Spare' | German: 'S3 966 Row 97 Spare Message German' | French: 'S3 966 Row 97 Spare Message French'
  967 = 'Spare' | German: 'S3 967 Row 97 Spare Message German' | French: 'S3 967 Row 97 Spare Message French'
  968 = 'Spare' | German: 'S3 968 Row 97 Spare Message German' | French: 'S3 968 Row 97 Spare Message French'
  969 = 'Spare' | German: 'S3 969 Row 97 Spare Message German' | French: 'S3 969 Row 97 Spare Message French'
  970 = 'Clamp Cylinder A1 Failed to Advance... Check Q1.0...' | German: 'S3 970 Row 98 Failed To Advance.. Check Qxxx.x German' | French: 'S3 970 Row 98 Failed To Advance.. Check Qxxx.x French'
  971 = 'Clamp Cylinder A1 Failed to Return... Check Q1.1...' | German: 'S3 971 Row 98 Failed To Return.. Check Qxxx.x German' | French: 'S3 971 Row 98 Failed To Return.. Check Qxxx.x French'
  972 = 'Clamp Cylinder A1 Lost Advanced... Check I1.0...' | German: 'S3 972 Row 98 Lost Advance Position... Check Ixxx.x German' | French: 'S3 972 Row 98 Lost Advance Position... Check Ixxx.x French'
  973 = 'Clamp Cylinder A1 Lost Returned... Check I1.1...' | German: 'S3 973 Row 98 Lost Return Position... Check Ixxx.x German' | French: 'S3 973 Row 98 Lost Return Position... Check Ixxx.x French'
  974 = 'Clamp Cylinder A1 Switch Fault... Check I1.0, I1.1...' | German: 'S3 974 Row 98 Switch Fault... Check Ixxx.x / Ixxx.x German' | French: 'S3 974 Row 98 Switch Fault... Check Ixxx.x / Ixxx.x French'
  975 = 'Spare' | German: 'S3 975 Row 98 Spare Message German' | French: 'S3 975 Row 98 Spare Message French'
  976 = 'Spare' | German: 'S3 976 Row 98 Spare Message German' | French: 'S3 976 Row 98 Spare Message French'
  977 = 'Spare' | German: 'S3 977 Row 98 Spare Message German' | French: 'S3 977 Row 98 Spare Message French'
  978 = 'Spare' | German: 'S3 978 Row 98 Spare Message German' | French: 'S3 978 Row 98 Spare Message French'
  979 = 'Spare' | German: 'S3 979 Row 98 Spare Message German' | French: 'S3 979 Row 98 Spare Message French'
  980 = 'Clamp Cylinder A1 Failed to Advance... Check Q1.0...' | German: 'S3 980 Row 99 Failed To Advance.. Check Qxxx.x German' | French: 'S3 980 Row 99 Failed To Advance.. Check Qxxx.x French'
  981 = 'Clamp Cylinder A1 Failed to Return... Check Q1.1...' | German: 'S3 981 Row 99 Failed To Return.. Check Qxxx.x German' | French: 'S3 981 Row 99 Failed To Return.. Check Qxxx.x French'
  982 = 'Clamp Cylinder A1 Lost Advanced... Check I1.0...' | German: 'S3 982 Row 99 Lost Advance Position... Check Ixxx.x German' | French: 'S3 982 Row 99 Lost Advance Position... Check Ixxx.x French'
  983 = 'Clamp Cylinder A1 Lost Returned... Check I1.1...' | German: 'S3 983 Row 99 Lost Return Position... Check Ixxx.x German' | French: 'S3 983 Row 99 Lost Return Position... Check Ixxx.x French'
  984 = 'Clamp Cylinder A1 Switch Fault... Check I1.0, I1.1...' | German: 'S3 984 Row 99 Switch Fault... Check Ixxx.x / Ixxx.x German' | French: 'S3 984 Row 99 Switch Fault... Check Ixxx.x / Ixxx.x French'
  985 = 'Spare' | German: 'S3 985 Row 99 Spare Message German' | French: 'S3 985 Row 99 Spare Message French'
  986 = 'Spare' | German: 'S3 986 Row 99 Spare Message German' | French: 'S3 986 Row 99 Spare Message French'
  987 = 'Spare' | German: 'S3 987 Row 99 Spare Message German' | French: 'S3 987 Row 99 Spare Message French'
  988 = 'Spare' | German: 'S3 988 Row 99 Spare Message German' | French: 'S3 988 Row 99 Spare Message French'
  989 = 'Spare' | German: 'S3 989 Row 99 Spare Message German' | French: 'S3 989 Row 99 Spare Message French'
  990 = 'S3 990 Row 100 Failed To Advance.. Check Qxxx.x Default' | German: 'S3 990 Row 100 Failed To Advance.. Check Qxxx.x German' | French: 'S3 990 Row 100 Failed To Advance.. Check Qxxx.x French'
  991 = 'S3 991 Row 100 Failed To Return.. Check Qxxx.x Default' | German: 'S3 991 Row 100 Failed To Return.. Check Qxxx.x German' | French: 'S3 991 Row 100 Failed To Return.. Check Qxxx.x French'
  992 = 'S3 992 Row 100 Lost Advance Position... Check Ixxx.x Default' | German: 'S3 992 Row 100 Lost Advance Position... Check Ixxx.x German' | French: 'S3 992 Row 100 Lost Advance Position... Check Ixxx.x French'
  993 = 'S3 993 Row 100 Lost Return Position... Check Ixxx.x Default' | German: 'S3 993 Row 100 Lost Return Position... Check Ixxx.x German' | French: 'S3 993 Row 100 Lost Return Position... Check Ixxx.x French'
  994 = 'S3 994 Row 100 Switch Fault... Check Ixxx.x / Ixxx.x Default' | German: 'S3 994 Row 100 Switch Fault... Check Ixxx.x / Ixxx.x German' | French: 'S3 994 Row 100 Switch Fault... Check Ixxx.x / Ixxx.x French'
  995 = 'S3 995 Row 100 Spare Message Default' | German: 'S3 995 Row 100 Spare Message German' | French: 'S3 995 Row 100 Spare Message French'
  996 = 'S3 996 Row 100 Spare Message Default' | German: 'S3 996 Row 100 Spare Message German' | French: 'S3 996 Row 100 Spare Message French'
  997 = 'S3 997 Row 100 Spare Message Default' | German: 'S3 997 Row 100 Spare Message German' | French: 'S3 997 Row 100 Spare Message French'
  998 = 'S3 998 Row 100 Spare Message Default' | German: 'S3 998 Row 100 Spare Message German' | French: 'S3 998 Row 100 Spare Message French'
  999 = 'S3 999 Row 100 Spare Message Default' | German: 'S3 999 Row 100 Spare Message German' | French: 'S3 999 Row 100 Spare Message French'
  1000 = 'S3_Alarms Default 1000' | German: 'S3_Alarms German 1000' | French: 'S3_Alarms French 1000'
   = ''
END_TEXTLIST

(* stored: Version 1.1.0.1, ProductVersion 3.1.4024.12
   TextList S3_Alarms: Id {f3fe854b-464f-4295-8a79-c774d357aaac} *)
